Fanuc KAREL source: kb00075.KL

-- PROVISIONAL review KL for V940-1; original PC SHA256 6d55e3d1c71bdd43126cf3f54c46af20471139d20b8888910f5fc30f32d3e1a4
-- Incomplete behavior may be omitted. Consult companion uncertainty JSON. Do not deploy.
PROGRAM KB00075
%NOLOCKGROUP
BEGIN
  -- V9_ZERO_TABLE_METADATA_HINT layout=0002_ascii; no indexed target words; source/name/runtime held
  -- UNRESOLVED_PC offsets 5-14; opcodes 3F,75
  -- UNRESOLVED_PC offsets 19-28; opcodes 3F,75
  -- UNRESOLVED_PC offsets 33-40; opcodes 9D,23
  -- UNRESOLVED_PC offsets 45-52; opcodes 9D,23
  -- UNRESOLVED_PC offsets 57-89; opcodes 27,22,2A,22,2A,22,22,31
  -- UNRESOLVED_PC offsets 94-98; opcodes 7F
END KB00075
